//{attribute 'qualified_only'}
//{attribute 'strict'}
TYPE E_DRIVE_DataType :
(*
Version history:
Date		|	Version/Author 		|	Remark
----------------------------------------------------------------------------------------------------
09.02.18	|	2.000.016	PSA		|	Original Version.
									|	Siemens G120 drive data type enumerations
*)
(
	//eNull, 
	//eBool, 
	//eInt, 
	//eDInt, 
	//eFloat
	eDUMMY
);
END_TYPE

(* stored: Version 1.1.0.1
   DUT E_DRIVE_DataType: Id {5154defd-8124-4f01-83cc-d926f80d061d} *)
